{attribute 'call_after_init'}
FUNCTION_BLOCK FINAL BoolParam EXTENDS BaseParam
VAR_INPUT
END_VAR
VAR_OUTPUT
	value: BOOL;
END_VAR
VAR
END_VAR

METHOD Change_Param
VAR_INPUT
	value	: STRING;
END_VAR
value := F_ToUCase(value);

IF value = '' OR value = '0' OR value = 'F' OR value = 'FALSE' OR value = 'OFF' THEN
	value := 'FALSE';
ELSE
	value := 'TRUE';
END_IF

THIS^.value := STRING_TO_BOOL(value);

IF THIS^.value THEN
	_display := 'ON';
ELSE
	_display := 'OFF';
END_IF
END_METHOD

METHOD Quick_Change
VAR_INPUT
	value: BOOL;
END_VAR
THIS^.value := value;

IF THIS^.value THEN
	_display := 'ON';
ELSE
	_display := 'OFF';
END_IF
END_METHOD

END_FUNCTION_BLOCK

(* stored: Version 1.1.0.1, ProductVersion 3.1.4024.12
   POU BoolParam: Id {2f01e2ae-9aef-46ce-80e0-d563f1f2ad2f}, SpecialFunc None
   Method Change_Param: Id {6e546fb4-4bcb-4897-9100-4ed85b8764c8}
   Method Quick_Change: Id {70185834-c71d-41c5-8e7a-1ad746e118f3} *)
